Staubli VAL3: SplitActionLine.pgx

public program SplitActionLine(string x_sLine, num& x_nDest[] (dimensions=3), num x_nFlag, bool& x_bRes)
  local num l_nData[25]
  local num l_nNum
  local num l_nBuff
  local string l_sChar[2]
begin

  x_bRes=false
  if x_sLine=="" or find(x_sLine,"=")<0
    return
  endIf

  x_sLine=right(x_sLine,len(x_sLine)-find(x_sLine,"=")-1)

  //如果这一行为空
  if x_sLine==""
    x_bRes=true
    return
  endIf


  //解析每一行
  l_sChar[0]=","
  l_sChar[1]=";"

  call SplitNumS(x_sLine,l_nData,l_sChar,x_bRes)

  if !x_bRes
    return
  endIf

  l_nBuff=0
  for l_nNum=0 to 11
    x_nDest[x_nFlag,l_nNum,0]=max(l_nData[l_nBuff],0)
    l_nBuff=l_nBuff+1
    x_nDest[x_nFlag,l_nNum,1]=max(l_nData[l_nBuff],0)
    l_nBuff=l_nBuff+1
  endFor





x_bRes=true






end
